(* PLC project Sin nombre, Desconocido Sin nombre 1 *)
(* stored: creationDateTime 2025-04-03T18:41:56, modificationDateTime 2025-04-07T16:46:15 *)

(* P_On *)
PROGRAM programBlink0
  VAR_INPUT RETAIN
    P_On : BOOL;
  END_VAR

(* LD diagram, written out as Structured Text *)
END_PROGRAM

CONFIGURATION Config0
  RESOURCE Res0 ON PLC
    TASK task0(INTERVAL := T#20ms, PRIORITY := 0);
    PROGRAM instance0 WITH task0 : programBlink0;
  END_RESOURCE
END_CONFIGURATION
